FUNCTION WRITE_PROTECTED_TIME
VAR_INPUT
    Ptr : POINTER TO TIME;
    Value : TIME;
END_VAR

Ptr^ := Value;

END_FUNCTION

(* stored: Version 1.1.0.1, ProductVersion 3.1.4022.18
   POU WRITE_PROTECTED_TIME: Id {fe63062b-7425-40a7-aecc-017a028de247}, SpecialFunc None *)
